TYPE ST_BaseComponent_HMI :
STRUCT
END_STRUCT
END_TYPE

(* stored: Version 1.1.0.1
   DUT ST_BaseComponent_HMI: Id {9a4adc48-322a-0770-2323-8e789531445d} *)
